FUNCTION_BLOCK COLOR_NAVY (* constant *)
  (* Standard: SO 11783-6 *)
  (* Version 1.0, 2022-07-29, franz *)
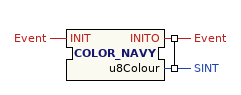
  EVENT_INPUT
    INIT; (* Service Initialization *)
  END_EVENT
  EVENT_OUTPUT
    INITO WITH u8Colour; (* Initialization Confirm *)
  END_EVENT
  VAR_OUTPUT
    u8Colour : SINT; (* Colour *)
  END_VAR
END_FUNCTION_BLOCK
